PROGRAM MAIN
VAR
	
	x1 : LREAL := -2;
	x2 : LREAL := 444;

	solution : ARRAY[0..7] OF LREAL;	

	fb_QPopt : Interface_TcCOM;
	
	TimeProfiler : Profiler;
END_VAR

TimeProfiler(START := TRUE, RESET := TRUE);

fb_QPopt.ip.solve(in1:= ADR(x1),  out1:= ADR(solution));

TimeProfiler(START := FALSE);

END_PROGRAM

(* stored: Version 1.1.0.1, ProductVersion 3.1.4024.12
   POU MAIN: Id {fd1777c2-2885-4a8f-bad3-bed6c970ef82}, SpecialFunc None *)
